TYPE HMIButtonMachineSection :
STRUCT
	IsEnabled	:	BOOL;
	IsPressed	:	BOOL;
	InPosition	:	BOOL;
	IsVisibleAxisPosition	:	BOOL;
	IsVisibleButton	:	BOOL;
	AxisPosition	:	REAL;
	CaptionButton	:	STRING;
	PathImageButton	:	STRING;
END_STRUCT
END_TYPE

(* stored: Version 1.1.0.1
   DUT HMIButtonMachineSection: Id {2ce3b5e1-29dd-491c-a6ff-4c55b64a6f27} *)
